// TIA Portal V20 export
DATA_BLOCK "BA010AZCR_ConveyorVirtualAxis"   // DB137, Motion_DB
// stored: InstanceOfName TO_SynchronousAxis, OfSystemLibElement TO_SynchronousAxis, OfSystemLibVersion 9.0
TO_SynchronousAxis   // technology object, version 9.0
// stored: SetPointCoupling Ref BA010AZCR_MasterVirtualAxis, Type TO_SynchronousAxis
   // // inherited from TO_PositioningAxis
   // // inherited from TO_SpeedAxis
   // // inherited from TO_Axis
   // // inherited from TO_Object
   // VAR
   //    Actor : TO_Struct_Actor;
   //    DynamicLimits : TO_Struct_DynamicLimits;
   //    DynamicDefaults : TO_Struct_DynamicDefaults;
   //    VirtualAxis : TO_Struct_VirtualAxis;
   // END_VAR
   // VAR
   //    Mechanics : TO_Struct_Mechanics;
   // END_VAR
   // VAR
   //    SynchronizedMotion { S7_SetPoint := 'True'} : TO_Struct_SynchronizedMotion;
   //    StatusSynchronizedMotion { ExternalWritable := 'False'; S7_SetPoint := 'True'} : TO_Struct_StatusSynchronizedMotion;
   // END_VAR
BEGIN
   Actor.DriveParameter.ReferenceSpeed := 8000.0;
   Actor.DriveParameter.MaxSpeed := 8000.0;
   DynamicLimits.MaxVelocity := 2000.0;
   DynamicLimits.MaxAcceleration := 40000.0;
   DynamicLimits.MaxDeceleration := 40000.0;
   DynamicLimits.MaxJerk := 800000.0;
   DynamicDefaults.EmergencyDeceleration := 40000.0;
   VirtualAxis.Mode := 1;
   Mechanics.LeadScrew := 15.0;
   VirtualAxis.Mode := 1;
END_DATA_BLOCK
